INTERFACE ITcoDialogAnswer EXTENDS ITcoDialogFormat

PROPERTY Answer : eDialogAnswer
GET
END_GET
END_PROPERTY

END_INTERFACE

(* stored: Version 1.1.0.1
   Itf ITcoDialogAnswer: Id {fe4969f0-7bd1-0730-1b30-bdd7ce347786}
   Property Answer: Id {334b806a-1dda-03c2-2fd2-78e87422dc63}
   Get Get: Id {e485c607-4df4-044c-341b-5a0d4d3fe2bc} *)
